Fanuc KAREL source: ko00001.KL

-- PROVISIONAL review KL for V1013-1; original PC SHA256 75aacd9e8189cb864d6bd5ed6bd43889bf497da0a4615e9bf282a4d312d39f24
-- Incomplete behavior may be omitted. Consult companion uncertainty JSON. Do not deploy.
PROGRAM KO00001
%NOLOCKGROUP
-- UNRESOLVED_DECL P1 type=000101
-- UNRESOLVED_DECL P2 type=000101
-- UNRESOLVED_DECL P3 type=000101
-- UNRESOLVED_DECL OUT type=000101
BEGIN
  -- UNRESOLVED_PC offsets 5-56; opcodes 27,22,1C,22,1C,22,1C,76,7E,4A
  -- UNRESOLVED_PC offsets 61-65; opcodes 7F
END KO00001
